PROGRAM JACK_CYCLE
VAR
END_VAR

jacks();

ACTION jacks:
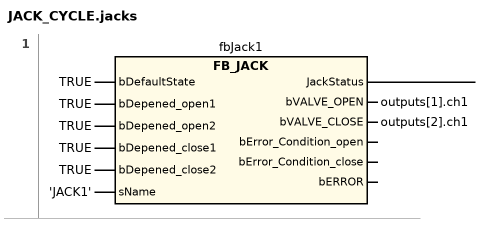
// NETWORK 1
fbJack1(
    bDefaultState := TRUE,
    bDepened_open1 := TRUE,
    bDepened_open2 := TRUE,
    bDepened_close1 := TRUE,
    bDepened_close2 := TRUE,
    sName := 'JACK1',
    bVALVE_OPEN => outputs[1].ch1,
    bVALVE_CLOSE => outputs[2].ch1); // FB_JACK
END_ACTION

END_PROGRAM

(* stored: Version 1.1.0.1, ProductVersion 3.1.4024.12
   POU JACK_CYCLE: Id {e77a0435-3511-4ef9-8780-98e171f4f5c1}, SpecialFunc None
   Action jacks: Id {3e047355-9a3b-462f-94b2-d42249bae2dc} *)
